(* PLC project FiveDofPlatform.project, CODESYS CODESYS V3.5 SP20 Patch 4 *)
(* stored: creationDateTime 2026-07-31T18:59:57.8348108, modificationDateTime 2026-07-31T18:56:30.8160222 *)

TYPE Axis : STRUCT
  Control_Mode : INT := 0;
  AxisEnable : BOOL;
  伺服绝对位置执行 : MC_MoveAbsolute;  (* 使用实际的功能块类型 *)
  AxisDone : BOOL;
  AxisBusy : BOOL;
  AxisError : BOOL;
  NeedMoveAxis : BOOL := FALSE;
  TargetVel : LREAL;
  TargetAngle : LREAL;
  TargetTorque : LREAL;
  ActualVel : LREAL;
  ActualAngle : LREAL;
  ActualTorque : LREAL;
  AxisLead : LREAL;
  AxisTravel : LREAL;
  AxisGearRatio : LREAL;
  InitDone : BOOL;
  TrigMove : INT;
  StopRequest : BOOL;
  AxisModeSwitchDone : BOOL;
END_STRUCT;
END_TYPE

TYPE LogEntry : STRUCT
  sMessage : STRING(100);  (* 日志内容 *)
  timestamp : DWORD;  (* 时间戳（例如毫秒） *)
  length : WORD;  (* 实际字符串长度 *)
END_STRUCT;
END_TYPE

TYPE LogBuffer : STRUCT
  entries : ARRAY[0..49] OF LogEntry;  (* 50条日志（索引0~49） *)
  writeIdx : INT;  (* 写入位置 (0~49) *)
  readIdx : INT;  (* 已读位置 *)
  count : INT;  (* 未读日志条数 (0~50) *)
  maxSize : INT := 50;  (* 缓冲区容量，固定50 *)
END_STRUCT;
END_TYPE

TYPE LogQueueEntry : STRUCT
  sMsg : STRING(100);
  timestamp : DWORD;
END_STRUCT;
END_TYPE

PROGRAM AxisStatusFeedback_PRG
  VAR
    fbStatusX : Sm3_Basic.MC_ReadStatus;
    fbAxisErrorX : Sm3_Basic.MC_ReadAxisError;
    fbStatusY : Sm3_Basic.MC_ReadStatus;
    fbAxisErrorY : Sm3_Basic.MC_ReadAxisError;
    fbStatusZ : Sm3_Basic.MC_ReadStatus;
    fbAxisErrorZ : Sm3_Basic.MC_ReadAxisError;
    fbStatusB : Sm3_Basic.MC_ReadStatus;
    fbAxisErrorB : Sm3_Basic.MC_ReadAxisError;
    fbStatusC : Sm3_Basic.MC_ReadStatus;
    fbAxisErrorC : Sm3_Basic.MC_ReadAxisError;
    wStatusX : WORD;
    wStatusY : WORD;
    wStatusZ : WORD;
    wStatusB : WORD;
    wStatusC : WORD;
    dwAxisErrorX : DWORD;
    dwAxisErrorY : DWORD;
    dwAxisErrorZ : DWORD;
    dwAxisErrorB : DWORD;
    dwAxisErrorC : DWORD;
    bStatusErrorX : BOOL;
    bStatusFBErrorX : BOOL;
    bStatusAxisErrorX : BOOL;
    bAxisErrorX : BOOL;
    bSwEndSwitchX : BOOL;
    bStatusErrorY : BOOL;
    bStatusFBErrorY : BOOL;
    bStatusAxisErrorY : BOOL;
    bAxisErrorY : BOOL;
    bSwEndSwitchY : BOOL;
    bStatusErrorZ : BOOL;
    bStatusFBErrorZ : BOOL;
    bStatusAxisErrorZ : BOOL;
    bAxisErrorZ : BOOL;
    bSwEndSwitchZ : BOOL;
    bStatusErrorB : BOOL;
    bStatusFBErrorB : BOOL;
    bStatusAxisErrorB : BOOL;
    bAxisErrorB : BOOL;
    bSwEndSwitchB : BOOL;
    bStatusErrorC : BOOL;
    bStatusFBErrorC : BOOL;
    bStatusAxisErrorC : BOOL;
    bAxisErrorC : BOOL;
    bSwEndSwitchC : BOOL;
  END_VAR

            
fbStatusX(
    Axis := AXIS_X,
    Enable := TRUE,
    Valid => ,
    Busy => ,
    Error => bStatusErrorX,
    ErrorID => ,
    Disabled => ,
    Errorstop => ,
    Stopping => ,
    StandStill => ,
    DiscreteMotion => ,
    ContinuousMotion => ,
    SynchronizedMotion => ,
    Homing => ,
    ConstantVelocity => ,
    Accelerating => ,
    Decelerating => ,
    FBErrorOccured => bStatusFBErrorX,
    AxisError => bStatusAxisErrorX
);

fbAxisErrorX(
    Axis := AXIS_X,
    Enable := TRUE,
    Valid => ,
    Busy => ,
    Error => ,
    ErrorID => ,
    AxisError => bAxisErrorX,
    AxisErrorID => dwAxisErrorX,
    SWEndSwitchActive => bSwEndSwitchX
);
IF NOT bAxisErrorX THEN
    dwAxisErrorX := DWORD#0;
END_IF;

wStatusX := WORD#0;
IF fbStatusX.Disabled THEN wStatusX := wStatusX OR WORD#16#0001; END_IF;
IF fbStatusX.Errorstop THEN wStatusX := wStatusX OR WORD#16#0002; END_IF;
IF fbStatusX.Stopping THEN wStatusX := wStatusX OR WORD#16#0004; END_IF;
IF fbStatusX.StandStill THEN wStatusX := wStatusX OR WORD#16#0008; END_IF;
IF fbStatusX.DiscreteMotion THEN wStatusX := wStatusX OR WORD#16#0010; END_IF;
IF fbStatusX.ContinuousMotion THEN wStatusX := wStatusX OR WORD#16#0020; END_IF;
IF fbStatusX.SynchronizedMotion THEN wStatusX := wStatusX OR WORD#16#0040; END_IF;
IF fbStatusX.Homing THEN wStatusX := wStatusX OR WORD#16#0080; END_IF;
IF fbStatusX.ConstantVelocity THEN wStatusX := wStatusX OR WORD#16#0100; END_IF;
IF fbStatusX.Accelerating THEN wStatusX := wStatusX OR WORD#16#0200; END_IF;
IF fbStatusX.Decelerating THEN wStatusX := wStatusX OR WORD#16#0400; END_IF;
IF bStatusErrorX THEN wStatusX := wStatusX OR WORD#16#0800; END_IF;
IF bStatusFBErrorX THEN wStatusX := wStatusX OR WORD#16#1000; END_IF;
IF bStatusAxisErrorX THEN wStatusX := wStatusX OR WORD#16#2000; END_IF;
IF bAxisErrorX THEN wStatusX := wStatusX OR WORD#16#4000; END_IF;
IF bSwEndSwitchX THEN wStatusX := wStatusX OR WORD#16#8000; END_IF;
arReg_data[16] := WORD_TO_INT(wStatusX);
arReg_data[22] := WORD_TO_INT(DWORD_TO_WORD(dwAxisErrorX));
arReg_data[23] := WORD_TO_INT(DWORD_TO_WORD(SHR(dwAxisErrorX, 16)));

fbStatusY(
    Axis := AXIS_Y,
    Enable := TRUE,
    Valid => ,
    Busy => ,
    Error => bStatusErrorY,
    ErrorID => ,
    Disabled => ,
    Errorstop => ,
    Stopping => ,
    StandStill => ,
    DiscreteMotion => ,
    ContinuousMotion => ,
    SynchronizedMotion => ,
    Homing => ,
    ConstantVelocity => ,
    Accelerating => ,
    Decelerating => ,
    FBErrorOccured => bStatusFBErrorY,
    AxisError => bStatusAxisErrorY
);

fbAxisErrorY(
    Axis := AXIS_Y,
    Enable := TRUE,
    Valid => ,
    Busy => ,
    Error => ,
    ErrorID => ,
    AxisError => bAxisErrorY,
    AxisErrorID => dwAxisErrorY,
    SWEndSwitchActive => bSwEndSwitchY
);
IF NOT bAxisErrorY THEN
    dwAxisErrorY := DWORD#0;
END_IF;

wStatusY := WORD#0;
IF fbStatusY.Disabled THEN wStatusY := wStatusY OR WORD#16#0001; END_IF;
IF fbStatusY.Errorstop THEN wStatusY := wStatusY OR WORD#16#0002; END_IF;
IF fbStatusY.Stopping THEN wStatusY := wStatusY OR WORD#16#0004; END_IF;
IF fbStatusY.StandStill THEN wStatusY := wStatusY OR WORD#16#0008; END_IF;
IF fbStatusY.DiscreteMotion THEN wStatusY := wStatusY OR WORD#16#0010; END_IF;
IF fbStatusY.ContinuousMotion THEN wStatusY := wStatusY OR WORD#16#0020; END_IF;
IF fbStatusY.SynchronizedMotion THEN wStatusY := wStatusY OR WORD#16#0040; END_IF;
IF fbStatusY.Homing THEN wStatusY := wStatusY OR WORD#16#0080; END_IF;
IF fbStatusY.ConstantVelocity THEN wStatusY := wStatusY OR WORD#16#0100; END_IF;
IF fbStatusY.Accelerating THEN wStatusY := wStatusY OR WORD#16#0200; END_IF;
IF fbStatusY.Decelerating THEN wStatusY := wStatusY OR WORD#16#0400; END_IF;
IF bStatusErrorY THEN wStatusY := wStatusY OR WORD#16#0800; END_IF;
IF bStatusFBErrorY THEN wStatusY := wStatusY OR WORD#16#1000; END_IF;
IF bStatusAxisErrorY THEN wStatusY := wStatusY OR WORD#16#2000; END_IF;
IF bAxisErrorY THEN wStatusY := wStatusY OR WORD#16#4000; END_IF;
IF bSwEndSwitchY THEN wStatusY := wStatusY OR WORD#16#8000; END_IF;
arReg_data[17] := WORD_TO_INT(wStatusY);
arReg_data[24] := WORD_TO_INT(DWORD_TO_WORD(dwAxisErrorY));
arReg_data[25] := WORD_TO_INT(DWORD_TO_WORD(SHR(dwAxisErrorY, 16)));

fbStatusZ(
    Axis := AXIS_Z,
    Enable := TRUE,
    Valid => ,
    Busy => ,
    Error => bStatusErrorZ,
    ErrorID => ,
    Disabled => ,
    Errorstop => ,
    Stopping => ,
    StandStill => ,
    DiscreteMotion => ,
    ContinuousMotion => ,
    SynchronizedMotion => ,
    Homing => ,
    ConstantVelocity => ,
    Accelerating => ,
    Decelerating => ,
    FBErrorOccured => bStatusFBErrorZ,
    AxisError => bStatusAxisErrorZ
);

fbAxisErrorZ(
    Axis := AXIS_Z,
    Enable := TRUE,
    Valid => ,
    Busy => ,
    Error => ,
    ErrorID => ,
    AxisError => bAxisErrorZ,
    AxisErrorID => dwAxisErrorZ,
    SWEndSwitchActive => bSwEndSwitchZ
);
IF NOT bAxisErrorZ THEN
    dwAxisErrorZ := DWORD#0;
END_IF;

wStatusZ := WORD#0;
IF fbStatusZ.Disabled THEN wStatusZ := wStatusZ OR WORD#16#0001; END_IF;
IF fbStatusZ.Errorstop THEN wStatusZ := wStatusZ OR WORD#16#0002; END_IF;
IF fbStatusZ.Stopping THEN wStatusZ := wStatusZ OR WORD#16#0004; END_IF;
IF fbStatusZ.StandStill THEN wStatusZ := wStatusZ OR WORD#16#0008; END_IF;
IF fbStatusZ.DiscreteMotion THEN wStatusZ := wStatusZ OR WORD#16#0010; END_IF;
IF fbStatusZ.ContinuousMotion THEN wStatusZ := wStatusZ OR WORD#16#0020; END_IF;
IF fbStatusZ.SynchronizedMotion THEN wStatusZ := wStatusZ OR WORD#16#0040; END_IF;
IF fbStatusZ.Homing THEN wStatusZ := wStatusZ OR WORD#16#0080; END_IF;
IF fbStatusZ.ConstantVelocity THEN wStatusZ := wStatusZ OR WORD#16#0100; END_IF;
IF fbStatusZ.Accelerating THEN wStatusZ := wStatusZ OR WORD#16#0200; END_IF;
IF fbStatusZ.Decelerating THEN wStatusZ := wStatusZ OR WORD#16#0400; END_IF;
IF bStatusErrorZ THEN wStatusZ := wStatusZ OR WORD#16#0800; END_IF;
IF bStatusFBErrorZ THEN wStatusZ := wStatusZ OR WORD#16#1000; END_IF;
IF bStatusAxisErrorZ THEN wStatusZ := wStatusZ OR WORD#16#2000; END_IF;
IF bAxisErrorZ THEN wStatusZ := wStatusZ OR WORD#16#4000; END_IF;
IF bSwEndSwitchZ THEN wStatusZ := wStatusZ OR WORD#16#8000; END_IF;
arReg_data[18] := WORD_TO_INT(wStatusZ);
arReg_data[26] := WORD_TO_INT(DWORD_TO_WORD(dwAxisErrorZ));
arReg_data[27] := WORD_TO_INT(DWORD_TO_WORD(SHR(dwAxisErrorZ, 16)));

fbStatusB(
    Axis := AXIS_B,
    Enable := TRUE,
    Valid => ,
    Busy => ,
    Error => bStatusErrorB,
    ErrorID => ,
    Disabled => ,
    Errorstop => ,
    Stopping => ,
    StandStill => ,
    DiscreteMotion => ,
    ContinuousMotion => ,
    SynchronizedMotion => ,
    Homing => ,
    ConstantVelocity => ,
    Accelerating => ,
    Decelerating => ,
    FBErrorOccured => bStatusFBErrorB,
    AxisError => bStatusAxisErrorB
);

fbAxisErrorB(
    Axis := AXIS_B,
    Enable := TRUE,
    Valid => ,
    Busy => ,
    Error => ,
    ErrorID => ,
    AxisError => bAxisErrorB,
    AxisErrorID => dwAxisErrorB,
    SWEndSwitchActive => bSwEndSwitchB
);
IF NOT bAxisErrorB THEN
    dwAxisErrorB := DWORD#0;
END_IF;

wStatusB := WORD#0;
IF fbStatusB.Disabled THEN wStatusB := wStatusB OR WORD#16#0001; END_IF;
IF fbStatusB.Errorstop THEN wStatusB := wStatusB OR WORD#16#0002; END_IF;
IF fbStatusB.Stopping THEN wStatusB := wStatusB OR WORD#16#0004; END_IF;
IF fbStatusB.StandStill THEN wStatusB := wStatusB OR WORD#16#0008; END_IF;
IF fbStatusB.DiscreteMotion THEN wStatusB := wStatusB OR WORD#16#0010; END_IF;
IF fbStatusB.ContinuousMotion THEN wStatusB := wStatusB OR WORD#16#0020; END_IF;
IF fbStatusB.SynchronizedMotion THEN wStatusB := wStatusB OR WORD#16#0040; END_IF;
IF fbStatusB.Homing THEN wStatusB := wStatusB OR WORD#16#0080; END_IF;
IF fbStatusB.ConstantVelocity THEN wStatusB := wStatusB OR WORD#16#0100; END_IF;
IF fbStatusB.Accelerating THEN wStatusB := wStatusB OR WORD#16#0200; END_IF;
IF fbStatusB.Decelerating THEN wStatusB := wStatusB OR WORD#16#0400; END_IF;
IF bStatusErrorB THEN wStatusB := wStatusB OR WORD#16#0800; END_IF;
IF bStatusFBErrorB THEN wStatusB := wStatusB OR WORD#16#1000; END_IF;
IF bStatusAxisErrorB THEN wStatusB := wStatusB OR WORD#16#2000; END_IF;
IF bAxisErrorB THEN wStatusB := wStatusB OR WORD#16#4000; END_IF;
IF bSwEndSwitchB THEN wStatusB := wStatusB OR WORD#16#8000; END_IF;
arReg_data[20] := WORD_TO_INT(wStatusB);
arReg_data[28] := WORD_TO_INT(DWORD_TO_WORD(dwAxisErrorB));
arReg_data[29] := WORD_TO_INT(DWORD_TO_WORD(SHR(dwAxisErrorB, 16)));

fbStatusC(
    Axis := AXIS_C,
    Enable := TRUE,
    Valid => ,
    Busy => ,
    Error => bStatusErrorC,
    ErrorID => ,
    Disabled => ,
    Errorstop => ,
    Stopping => ,
    StandStill => ,
    DiscreteMotion => ,
    ContinuousMotion => ,
    SynchronizedMotion => ,
    Homing => ,
    ConstantVelocity => ,
    Accelerating => ,
    Decelerating => ,
    FBErrorOccured => bStatusFBErrorC,
    AxisError => bStatusAxisErrorC
);

fbAxisErrorC(
    Axis := AXIS_C,
    Enable := TRUE,
    Valid => ,
    Busy => ,
    Error => ,
    ErrorID => ,
    AxisError => bAxisErrorC,
    AxisErrorID => dwAxisErrorC,
    SWEndSwitchActive => bSwEndSwitchC
);
IF NOT bAxisErrorC THEN
    dwAxisErrorC := DWORD#0;
END_IF;

wStatusC := WORD#0;
IF fbStatusC.Disabled THEN wStatusC := wStatusC OR WORD#16#0001; END_IF;
IF fbStatusC.Errorstop THEN wStatusC := wStatusC OR WORD#16#0002; END_IF;
IF fbStatusC.Stopping THEN wStatusC := wStatusC OR WORD#16#0004; END_IF;
IF fbStatusC.StandStill THEN wStatusC := wStatusC OR WORD#16#0008; END_IF;
IF fbStatusC.DiscreteMotion THEN wStatusC := wStatusC OR WORD#16#0010; END_IF;
IF fbStatusC.ContinuousMotion THEN wStatusC := wStatusC OR WORD#16#0020; END_IF;
IF fbStatusC.SynchronizedMotion THEN wStatusC := wStatusC OR WORD#16#0040; END_IF;
IF fbStatusC.Homing THEN wStatusC := wStatusC OR WORD#16#0080; END_IF;
IF fbStatusC.ConstantVelocity THEN wStatusC := wStatusC OR WORD#16#0100; END_IF;
IF fbStatusC.Accelerating THEN wStatusC := wStatusC OR WORD#16#0200; END_IF;
IF fbStatusC.Decelerating THEN wStatusC := wStatusC OR WORD#16#0400; END_IF;
IF bStatusErrorC THEN wStatusC := wStatusC OR WORD#16#0800; END_IF;
IF bStatusFBErrorC THEN wStatusC := wStatusC OR WORD#16#1000; END_IF;
IF bStatusAxisErrorC THEN wStatusC := wStatusC OR WORD#16#2000; END_IF;
IF bAxisErrorC THEN wStatusC := wStatusC OR WORD#16#4000; END_IF;
IF bSwEndSwitchC THEN wStatusC := wStatusC OR WORD#16#8000; END_IF;
arReg_data[21] := WORD_TO_INT(wStatusC);
arReg_data[30] := WORD_TO_INT(DWORD_TO_WORD(dwAxisErrorC));
arReg_data[31] := WORD_TO_INT(DWORD_TO_WORD(SHR(dwAxisErrorC, 16)));
            
          
END_PROGRAM

PROGRAM Axis_Y_PRG
  VAR
    伺服使能 : Sm3_Basic.MC_Power;  (* 轴功能块实例 *)
    伺服绝对位置执行 : Sm3_Basic.MC_MoveAbsolute;
    伺服实际位置 : Sm3_Basic.MC_ReadActualPosition;
    伺服停止 : Sm3_Basic.MC_Stop;
    伺服复位 : Sm3_Basic.MC_Reset;
    伺服状态 : Sm3_Basic.MC_ReadStatus;
    复位轴组 : Sm3_Basic.SMC3_ReinitDrive;
    当前位置 : LREAL;  (* 变量 *)
    轴组复位 : BOOL;
    目标位置 : LREAL;
    目标速度 : LREAL;
    伺服错误状态 : BOOL;
    轴使能状态 : BOOL;
    总线状态 : BOOL;
    复位触发 : R_TRIG;  (* 报警清除相关 *)
    复位请求 : BOOL;
    复位中 : BOOL;
    POS_DEAD_ZONE : REAL := 0.01;  (* 死区常量 *)
    伺服复位_Done : BOOL;
    debug_Done_Status : BOOL;  (* 在 AXIS_Y0_PRG 中添加 *)
    debug_KeepEnable : BOOL;
    move_trigger : R_TRIG;  (* 脉冲触发相关 *)
    AXIS_Y_EXCUSE : BOOL := FALSE;
    log_msg : STRING(100);
  END_VAR

                    //------------------------------------------------------------------
// Z 轴控制逻辑（简化版 - 仅上升沿触发）
//------------------------------------------------------------------

// 读取实际位置
伺服实际位置(
    Axis    := AXIS_Y,
    Enable  := TRUE,
    Position=> 当前位置
);
GVL.Axes[2].ActualAngle := 当前位置;

// 读取轴状态
伺服状态(
    Axis    := AXIS_Y,
    Enable  := TRUE,
    Valid   => ,
    Busy    => ,
    Error   => 伺服错误状态,
    ErrorID => ,
    Disabled=> 总线状态
);

// 轴使能控制
伺服使能(
    Axis               := AXIS_Y,
    Enable             := TRUE,
    bRegulatorOn       := GVL.Axes[2].AxisEnable,
    bDriveStart        := GVL.Axes[2].AxisEnable,
    Status             => 轴使能状态,
    bRegulatorRealState=> ,
    bDriveStartRealState=> ,
    Busy               => ,
    Error              => ,
    ErrorID            =>
);

// 目标位置、速度赋值（来自全局变量）
目标位置 := GVL.Axes[2].TargetAngle;
目标速度 :=  GVL.Axes[2].TargetVel;

// ********** 核心：上升沿触发运动 **********
// 使用 R_TRIG 检测 need_move 的上升沿
move_trigger(CLK := GVL.Axes[2].NeedMoveAxis);
IF move_trigger.Q THEN
    AXIS_Y_EXCUSE := TRUE;   // 产生一个扫描周期的脉冲
	log_msg := 'X-axis has been triggered';
// 	logfb(write:=TRUE,sFileTestString:=log_msg);
	AppendLog(log_msg);
ELSE
    AXIS_Y_EXCUSE := FALSE;
END_IF

// 绝对定位指令
GVL.Axes[2].伺服绝对位置执行(
    Axis        := AXIS_Y,
    Execute     := AXIS_Y_EXCUSE,
    Position    := 目标位置,
    Velocity    := 目标速度,
    Acceleration:= 10000,//4000  //85000
    Deceleration:= 10000,//4000  //85000
    Jerk        := ,
    Direction   := ,
    BufferMode  := ,
    Done        => GVL.Axes[2].InitDone,
    Busy        => ,
    Active      => ,
    CommandAborted=> ,
    Error       => GVL.Axes[2].AxisError,
    ErrorID     =>
);

// 运动完成：清除 need_move 并通知状态机
IF  GVL.Axes[2].InitDone THEN
    GVL.Axes[2].NeedMoveAxis := FALSE;              // 清除运动请求
    GVL.Axes[2].AxisDone := TRUE;         // 通知状态机运动完成
	log_msg := 'X-Axis movement completed! ';
// 	logfb(write:=TRUE,sFileTestString:=log_msg);
// 	AppendLog(log_msg);
END_IF

// 复位功能块（保持不变）
伺服复位(
    Axis    := AXIS_Y,
    Execute := 复位中 AND NOT 伺服复位.Done,
    Done    => ,
    Busy    => ,
    Error   => ,
    ErrorID =>
);

复位轴组(
    Axis      := AXIS_Y,
    bExecute  := 伺服复位.Done,
    bVirtual  := FALSE,
    bDone     => ,
    bBusy     => ,
    bError    => ,
    nErrorID  =>
);

// 报警清除逻辑
复位触发(CLK := (伺服错误状态 OR 复位请求) AND NOT 复位中);
IF 复位触发.Q THEN
    复位中 := TRUE;
    复位请求 := FALSE;
END_IF

IF 伺服复位.Done THEN
    复位中 := FALSE;
END_IF
                  
END_PROGRAM

PROGRAM ModbusTcpSlave
  VAR CONSTANT
    aAngleFactor : ARRAY[1..GVL.AXIS_COUNT] OF REAL := [(360.0 / 26.0), (360.0 / 5.0), (360.0 / 5.0), 1, 1];
  END_VAR
  VAR
    modTcpSlaveInit : gcan.FB_ModbusTCP_Slave_Init;  (* Modbus TCP Slave初始化功能块 *)
    modTcpSlaveCtrl : gcan.FB_ModbusTCP_Slave_Ctrl;  (* Modbus TCP Slave执行功能块 *)
    eout : BOOL;  (* 用于承接功能块中完成标志引脚数据的变量 *)
    iSocket : INT;  (* 用于存放自身socket *)
    uiErr : UINT;  (* 用于承接功能块中报错引脚错误信息的变量 *)
    isInit : BOOL := FALSE;  (* 用于初始化执行一次的逻辑变量 *)
    arClient : ARRAY[0..10] OF INT;  (* 用于存放Client即主站的socket *)
    btargetAngleChange : BOOL := FALSE;
    OldTargetAngle : WORD;
    enCtr : BOOL := FALSE;  (* Modbus TCP Slave执行功能块使能变量 *)
    iTemp : INT;  (* 临时变量，用于32位数据转换 *)
    dwAngle : INT;  (* 32位临时存储，用于组合角度寄存器 *)
    i : INT;
    wTemp : WORD;  (* modbuslog *)
    sCurLog : STRING(100);
    iLen : INT;
    pCurEntry : POINTER TO LogEntry;
    iCharIdx : INT;
    iRegIdx : INT;
  END_VAR

                    // ================================
// 日志映射部分：将当前未读日志填充到保持寄存器
// ================================
IF g_LogBuffer.count > 0 THEN
    // 获取当前读指针指向的日志条目
    pCurEntry := ADR(g_LogBuffer.entries[g_LogBuffer.readIdx]);
    sCurLog := pCurEntry^.sMessage;
    iLen := pCurEntry^.length;
    
    // 地址100：日志长度（WORD）
    arReg_data[100] := INT_TO_WORD(iLen);
    
    // 地址101-102：时间戳（低字，高字）
    arReg_data[101] := DWORD_TO_WORD(pCurEntry^.timestamp AND 16#FFFF);
    arReg_data[102] := DWORD_TO_WORD(SHR(pCurEntry^.timestamp, 16));
    
    // 清空字符串缓冲区寄存器（地址103 ~ 152，共50个WORD）
    FOR i := 103 TO 152 DO
        arReg_data[i] := 0;
    END_FOR
    
    // ----- 将字符串每两个字符打包成一个 WORD -----
    // 注意：你的环境中字符串索引从0开始（已验证）
    iCharIdx := 0;      // 当前字符索引（从0开始）
    iRegIdx := 103;     // 当前寄存器地址
    WHILE iCharIdx < iLen DO
        // 低字节 = 第一个字符
        wTemp := sCurLog[iCharIdx];
        iCharIdx := iCharIdx + 1;
        // 如果有下一个字符，放入高字节
        IF iCharIdx < iLen THEN
            wTemp := wTemp OR SHL(sCurLog[iCharIdx], 8);
            iCharIdx := iCharIdx + 1;
        END_IF
        arReg_data[iRegIdx] := wTemp;
        iRegIdx := iRegIdx + 1;
    END_WHILE
ELSE
    // 无未读日志，长度寄存器写0
    arReg_data[100] := 0;
END_IF

// --------------------------------
// 处理主站确认线圈（地址16）
// --------------------------------
IF arDo_data[16] THEN
    IF g_LogBuffer.count > 0 THEN
        g_LogBuffer.readIdx := (g_LogBuffer.readIdx + 1) MOD g_LogBuffer.maxSize;
        g_LogBuffer.count := g_LogBuffer.count - 1;
    END_IF
    arDo_data[16] := FALSE;
END_IF





IF isInit=FALSE THEN							

	modtcpslaveinit(en_in:=TRUE,					//Modbus TCP Slave初始化功能块使能
	xenable:=TRUE,									//使能初始化功能
	iport:=502,										//开放端口号502
	en_out=>eout,									//Modbus TCP Slave初始化功能块执行完成
	isocket=>iSocket,								//创建的socket存入变量
	uierror=>uiErr);								//Modbus TCP Slave初始化功能块执行错误信息
	
	IF isocket>=0 AND uiErr=0 THEN					//成功创建socket且无错误，逻辑标志置位，下周期执行ELSE
		isInit:=TRUE;	
		
		enCtr:=FALSE;
		ELSE                                        //等待连接成功
		modtcpslaveinit(en_in:=0,xenable:=0);	
	END_IF
 
ELSE


	// 循环读取电机位置
	FOR i := 1 TO GVL.AXIS_COUNT DO
		arAi_data[i] := INT_TO_WORD(REAL_TO_INT(Axes[i].ActualAngle/aAngleFactor[i]*10.0));
	END_FOR
	Move_5Axis_Sign:=arReg_data[0];
	
	
	// 循环处理前7个通道（目标角度数组）
	IF 	bfiveDOF_state =0 THEN
		FOR i := 1 TO GVL.AXIS_COUNT DO
			dwAngle := WORD_TO_INT(arReg_data[i]);      // 有符号原始值
			PlatformTargetAngle[i] := dwAngle * aAngleFactor[i];
		END_FOR

	END_IF
  xJogMode[1] := (arReg_data[19] AND WORD#16#0001) <> WORD#0; // X
  xJogMode[2] := (arReg_data[19] AND WORD#16#0002) <> WORD#0; // Y
  xJogMode[3] := (arReg_data[19] AND WORD#16#0004) <> WORD#0; // Z
  xJogMode[4] := (arReg_data[19] AND WORD#16#0008) <> WORD#0; // B
  xJogMode[5] := (arReg_data[19] AND WORD#16#0010) <> WORD#0; // C
  
  xJogFwd[1] := xJogMode[1] AND (arReg_data[6] <> WORD#0);
  xJogRev[1] := xJogMode[1] AND (arReg_data[7] <> WORD#0);

  xJogFwd[2] := xJogMode[2] AND (arReg_data[8] <> WORD#0);
  xJogRev[2] := xJogMode[2] AND (arReg_data[9] <> WORD#0);

  xJogFwd[3] := xJogMode[3] AND (arReg_data[10] <> WORD#0);
  xJogRev[3] := xJogMode[3] AND (arReg_data[11] <> WORD#0);

  xJogFwd[4] := xJogMode[4] AND (arReg_data[12] <> WORD#0);
  xJogRev[4] := xJogMode[4] AND (arReg_data[13] <> WORD#0);

  xJogFwd[5] := xJogMode[5] AND (arReg_data[14] <> WORD#0);
  xJogRev[5] := xJogMode[5] AND (arReg_data[15] <> WORD#0);
  
  xJogFwd[1] := arReg_data[6] <> 0;
  xJogRev[1] := arReg_data[7] <> 0;

  xJogFwd[2] := arReg_data[8] <> 0;
  xJogRev[2] := arReg_data[9] <> 0;

  xJogFwd[3] := arReg_data[10] <> 0;
  xJogRev[3] := arReg_data[11] <> 0;

  xJogFwd[4] := arReg_data[12] <> 0;
  xJogRev[4] := arReg_data[13] <> 0;

  xJogFwd[5] := arReg_data[14] <> 0;
  xJogRev[5] := arReg_data[15] <> 0;

	modtcpslavectrl(en_in:=enCtr,					//Modbus TCP Slave执行功能块使能
	xenable:=TRUE,									//Modbus TCP Slave执行功能使能
	isocket:=isocket,								//输入创建的socket
	dwatchdogtime:=2000,							//看门狗时间
	p_clientsocket:=ADR(arClient),					//将连接进来的socket存放到数组
	imaxclientcount:=10,							//设置最大连接数量
	uido_number:=17,uido_startaddr:=0,pdo_data:=ADR(arDo_data),		//uido_number设定线圈个数，uido_startaddr设定线圈起始地址，数据存放在arDo_data数组
	uidi_number:=16,uidi_startaddr:=0,pdi_data:=ADR(arDi_data),		//uidi_number设定离散型数据个数，uidi_startaddr设定离散型数据起始地址，数据存放在arDi_data数组
	uireg_number:=200,uireg_startaddr:=0,preg_data:=ADR(arReg_data), //uireg_number设定保持型寄存器个数，uireg_startaddr设定保持型寄存器起始地址，数据存放在arReg_data数组
	uiai_number:=16,uiai_startaddr:=0,pai_data:=ADR(arAi_data),		//uiai_number设定输入型寄存器个数，uiai_startaddr设定输入型寄存器起始地址，数据存放在arAi_data数组
	en_out=>eout,									//Modbus TCP Slave执行功能块执行完成
	uierror=>uierr);								//Modbus TCP Slave执行功能块执行错误信息
	enctr:=TRUE;
	IF uierr <>0 THEN                               //如果从站报错，则重新连接从站
		modtcpslaveinit(en_in:=0,xenable:=0);	
		isInit:=0;
	END_IF
END_IF

 
// 释放锁
g_LogLock := FALSE;
 
                  
END_PROGRAM

PROGRAM PLC_PRG
  VAR
    startMove : BOOL;
    platTargetangle : ARRAY[1..7] OF LREAL;
    platTargetvel : ARRAY[1..7] OF LREAL;
    fbMove6DOF : FB_5DOF_Platform_Move;
    iAxis : INT;
    MaxVel : UDINT := 2048576000;
    bcontrol : UINT;
    logfb : Syslog_FB;
    log_msg : STRING(100);
  END_VAR

                    
                  
END_PROGRAM

FUNCTION_BLOCK FB_5DOF_Platform_Move
  VAR_IN_OUT
    AxisAngle : ARRAY[1..AXIS_COUNT] OF LREAL;
    AxisVel : ARRAY[1..AXIS_COUNT] OF LREAL;
  END_VAR
  VAR_INPUT
    Execute : BOOL;
    Monitor : BOOL;
  END_VAR
  VAR_OUTPUT
    Done : BOOL;
    Busy : BOOL;
    Error : BOOL;
    ErrorID : WORD;
  END_VAR
  VAR
    trigExec : R_TRIG;
    xInternal : BOOL;
    i : INT;
    allDone : BOOL := FALSE;
    anyError : BOOL;
    errId : WORD;
  END_VAR

                    
// 上升沿触发：锁存目标值并开始运动
trigExec(CLK := Execute);
IF trigExec.Q THEN
    FOR i := 1 TO AXIS_COUNT DO
        GVL.Axes[i].TargetAngle := AxisAngle[i];
		GVL.Axes[i].TargetVel:=AxisVel[i];
    END_FOR
//     xInternal := TRUE;
    Busy := TRUE;
    Done := FALSE;
    Error := FALSE;
    ErrorID := 0;
END_IF

// 监控所有轴的状态（需要你的单轴功能块实例：AXIS_X伺服绝对位置执行 等）
IF Monitor  THEN
    allDone := TRUE;
    anyError := FALSE;
    errId := 0;
    
    // 检查每个轴（请根据实际轴名修改，以下为示例）
	FOR i :=1 TO AXIS_COUNT DO
		IF NOT GVL.Axes[i].AxisDone THEN allDone := FALSE; END_IF
		IF GVL.Axes[i].AxisError THEN anyError := TRUE; errId := GVL.Axes[i].伺服绝对位置执行.ErrorID; END_IF
	END_FOR
  
    
    IF  allDone THEN
        Busy := FALSE;
        Done := TRUE;
        xInternal := FALSE;
    END_IF
END_IF
                  
END_FUNCTION_BLOCK

PROGRAM AXIS_X_PRG
  VAR
    伺服使能 : Sm3_Basic.MC_Power;  (* 轴功能块实例 *)
    伺服绝对位置执行 : Sm3_Basic.MC_MoveAbsolute;
    伺服实际位置 : Sm3_Basic.MC_ReadActualPosition;
    伺服停止 : Sm3_Basic.MC_Stop;
    伺服复位 : Sm3_Basic.MC_Reset;
    伺服状态 : Sm3_Basic.MC_ReadStatus;
    复位轴组 : Sm3_Basic.SMC3_ReinitDrive;
    当前位置 : LREAL;  (* 变量 *)
    轴组复位 : BOOL;
    目标位置 : LREAL;
    目标速度 : LREAL;
    伺服错误状态 : BOOL;
    轴使能状态 : BOOL;
    总线状态 : BOOL;
    复位触发 : R_TRIG;  (* 报警清除相关 *)
    复位请求 : BOOL;
    复位中 : BOOL;
    POS_DEAD_ZONE : REAL := 0.01;  (* 死区常量 *)
    move_trigger : R_TRIG;
    AXIS_X_EXCUSE : BOOL := FALSE;
    log_msg : STRING(100);
  END_VAR

                    //------------------------------------------------------------------
// Z 轴控制逻辑（简化版 - 仅上升沿触发）
//------------------------------------------------------------------

// 读取实际位置
伺服实际位置(
    Axis    := AXIS_X,
    Enable  := TRUE,
    Position=> 当前位置
);
GVL.Axes[1].ActualAngle := 当前位置;

// 读取轴状态
伺服状态(
    Axis    := AXIS_X,
    Enable  := TRUE,
    Valid   => ,
    Busy    => ,
    Error   => 伺服错误状态,
    ErrorID => ,
    Disabled=> 总线状态
);

// 轴使能控制
伺服使能(
    Axis               := AXIS_X,
    Enable             := TRUE,
    bRegulatorOn       := GVL.Axes[1].AxisEnable,
    bDriveStart        := GVL.Axes[1].AxisEnable,
    Status             => 轴使能状态,
    bRegulatorRealState=> ,
    bDriveStartRealState=> ,
    Busy               => ,
    Error              => ,
    ErrorID            =>
);

// 目标位置、速度赋值（来自全局变量）
目标位置 := GVL.Axes[1].TargetAngle;
目标速度 :=  GVL.Axes[1].TargetVel;

// ********** 核心：上升沿触发运动 **********
// 使用 R_TRIG 检测 need_move 的上升沿
move_trigger(CLK := GVL.Axes[1].NeedMoveAxis);
IF move_trigger.Q THEN
    AXIS_X_EXCUSE := TRUE;   // 产生一个扫描周期的脉冲
	log_msg := 'X-axis has been triggered';
// 	logfb(write:=TRUE,sFileTestString:=log_msg);
	AppendLog(log_msg);
ELSE
    AXIS_X_EXCUSE := FALSE;
END_IF

// 绝对定位指令
GVL.Axes[1].伺服绝对位置执行(
    Axis        := AXIS_X,
    Execute     := AXIS_X_EXCUSE,
    Position    := 目标位置,
    Velocity    := 目标速度,
    Acceleration:= 10000,//4000  //85000
    Deceleration:= 10000,//4000  //85000
    Jerk        := ,
    Direction   := ,
    BufferMode  := ,
    Done        => GVL.Axes[1].InitDone,
    Busy        => ,
    Active      => ,
    CommandAborted=> ,
    Error       => GVL.Axes[1].AxisError,
    ErrorID     =>
);

// 运动完成：清除 need_move 并通知状态机
IF  GVL.Axes[1].InitDone THEN
    GVL.Axes[1].NeedMoveAxis := FALSE;              // 清除运动请求
    GVL.Axes[1].AxisDone := TRUE;         // 通知状态机运动完成
	log_msg := 'X-Axis movement completed! ';
// 	logfb(write:=TRUE,sFileTestString:=log_msg);
// 	AppendLog(log_msg);
END_IF

// 复位功能块（保持不变）
伺服复位(
    Axis    := AXIS_X,
    Execute := 复位中 AND NOT 伺服复位.Done,
    Done    => ,
    Busy    => ,
    Error   => ,
    ErrorID =>
);

复位轴组(
    Axis      := AXIS_X,
    bExecute  := 伺服复位.Done,
    bVirtual  := FALSE,
    bDone     => ,
    bBusy     => ,
    bError    => ,
    nErrorID  =>
);

// 报警清除逻辑
复位触发(CLK := (伺服错误状态 OR 复位请求) AND NOT 复位中);
IF 复位触发.Q THEN
    复位中 := TRUE;
    复位请求 := FALSE;
END_IF

IF 伺服复位.Done THEN
    复位中 := FALSE;
END_IF
                  
END_PROGRAM

PROGRAM AXIS_B_PRG
  VAR
    伺服使能 : Sm3_Basic.MC_Power;  (* 轴功能块实例 *)
    伺服绝对位置执行 : Sm3_Basic.MC_MoveAbsolute;
    伺服实际位置 : Sm3_Basic.MC_ReadActualPosition;
    伺服停止 : Sm3_Basic.MC_Stop;
    伺服复位 : Sm3_Basic.MC_Reset;
    伺服状态 : Sm3_Basic.MC_ReadStatus;
    复位轴组 : Sm3_Basic.SMC3_ReinitDrive;
    当前位置 : LREAL;  (* 变量 *)
    轴组复位 : BOOL;
    目标位置 : LREAL;
    目标速度 : LREAL;
    伺服错误状态 : BOOL;
    轴使能状态 : BOOL;
    总线状态 : BOOL;
    复位触发 : R_TRIG;  (* 报警清除相关 *)
    复位请求 : BOOL;
    复位中 : BOOL;
    move_trigger : R_TRIG;
    AXIS_B_EXCUSE : BOOL := FALSE;
    log_msg : STRING(100);
  END_VAR

                    //------------------------------------------------------------------
// Z 轴控制逻辑（简化版 - 仅上升沿触发）
//------------------------------------------------------------------

// 读取实际位置
伺服实际位置(
    Axis    := AXIS_B,
    Enable  := TRUE,
    Position=> 当前位置
);
GVL.Axes[4].ActualAngle := 当前位置;

// 读取轴状态
伺服状态(
    Axis    := AXIS_B,
    Enable  := TRUE,
    Valid   => ,
    Busy    => ,
    Error   => 伺服错误状态,
    ErrorID => ,
    Disabled=> 总线状态
);

// 轴使能控制
伺服使能(
    Axis               := AXIS_B,
    Enable             := TRUE,
    bRegulatorOn       := GVL.Axes[4].AxisEnable,
    bDriveStart        := GVL.Axes[4].AxisEnable,
    Status             => 轴使能状态,
    bRegulatorRealState=> ,
    bDriveStartRealState=> ,
    Busy               => ,
    Error              => ,
    ErrorID            =>
);

// 目标位置、速度赋值（来自全局变量）
目标位置 := GVL.Axes[4].TargetAngle;
目标速度 :=  GVL.Axes[4].TargetVel;

// ********** 核心：上升沿触发运动 **********
// 使用 R_TRIG 检测 need_move 的上升沿
move_trigger(CLK := GVL.Axes[4].NeedMoveAxis);
IF move_trigger.Q THEN
    AXIS_B_EXCUSE := TRUE;   // 产生一个扫描周期的脉冲
	log_msg := 'X-axis has been triggered';
// 	logfb(write:=TRUE,sFileTestString:=log_msg);
	AppendLog(log_msg);
ELSE
    AXIS_B_EXCUSE := FALSE;
END_IF

// 绝对定位指令
GVL.Axes[4].伺服绝对位置执行(
    Axis        := AXIS_B,
    Execute     := AXIS_B_EXCUSE,
    Position    := 目标位置,
    Velocity    := 目标速度,
    Acceleration:= 10000,//4000  //85000
    Deceleration:= 10000,//4000  //85000
    Jerk        := ,
    Direction   := ,
    BufferMode  := ,
    Done        => GVL.Axes[4].InitDone,
    Busy        => ,
    Active      => ,
    CommandAborted=> ,
    Error       => GVL.Axes[4].AxisError,
    ErrorID     =>
);

// 运动完成：清除 need_move 并通知状态机
IF  GVL.Axes[4].InitDone THEN
    GVL.Axes[4].NeedMoveAxis := FALSE;              // 清除运动请求
    GVL.Axes[4].AxisDone := TRUE;         // 通知状态机运动完成
	log_msg := 'B-Axis movement completed! ';
// 	logfb(write:=TRUE,sFileTestString:=log_msg);
// 	AppendLog(log_msg);
END_IF

// 复位功能块（保持不变）
伺服复位(
    Axis    := AXIS_B,
    Execute := 复位中 AND NOT 伺服复位.Done,
    Done    => ,
    Busy    => ,
    Error   => ,
    ErrorID =>
);

复位轴组(
    Axis      := AXIS_B,
    bExecute  := 伺服复位.Done,
    bVirtual  := FALSE,
    bDone     => ,
    bBusy     => ,
    bError    => ,
    nErrorID  =>
);

// 报警清除逻辑
复位触发(CLK := (伺服错误状态 OR 复位请求) AND NOT 复位中);
IF 复位触发.Q THEN
    复位中 := TRUE;
    复位请求 := FALSE;
END_IF

IF 伺服复位.Done THEN
    复位中 := FALSE;
END_IF
                  
END_PROGRAM

PROGRAM AXIS_Z_PRG
  VAR
    伺服使能 : Sm3_Basic.MC_Power;  (* 轴功能块实例 *)
    伺服绝对位置执行 : Sm3_Basic.MC_MoveAbsolute;
    伺服实际位置 : Sm3_Basic.MC_ReadActualPosition;
    伺服停止 : Sm3_Basic.MC_Stop;
    伺服复位 : Sm3_Basic.MC_Reset;
    伺服状态 : Sm3_Basic.MC_ReadStatus;
    复位轴组 : Sm3_Basic.SMC3_ReinitDrive;
    当前位置 : LREAL;  (* 变量 *)
    轴组复位 : BOOL;
    目标位置 : LREAL;
    目标速度 : LREAL;
    伺服错误状态 : BOOL;
    轴使能状态 : BOOL;
    总线状态 : BOOL;
    复位触发 : R_TRIG;  (* 报警清除相关 *)
    复位请求 : BOOL;
    复位中 : BOOL;
    伺服复位_Done : BOOL;
    debug_Done_Status : BOOL;  (* 在 AXIS_Z_PRG 中添加 *)
    debug_KeepEnable : BOOL;
    move_trigger : R_TRIG;  (* 脉冲触发相关 *)
    AXIS_Z_EXCUSE : BOOL := FALSE;
    log_msg : STRING(100);
  END_VAR

                    //------------------------------------------------------------------
// Z 轴控制逻辑（简化版 - 仅上升沿触发）
//------------------------------------------------------------------

// 读取实际位置
伺服实际位置(
    Axis    := AXIS_Z,
    Enable  := TRUE,
    Position=> 当前位置
);
GVL.Axes[3].ActualAngle := 当前位置;

// 读取轴状态
伺服状态(
    Axis    := AXIS_Z,
    Enable  := TRUE,
    Valid   => ,
    Busy    => ,
    Error   => 伺服错误状态,
    ErrorID => ,
    Disabled=> 总线状态
);

// 轴使能控制
伺服使能(
    Axis               := AXIS_Z,
    Enable             := TRUE,
    bRegulatorOn       := GVL.Axes[3].AxisEnable,
    bDriveStart        := GVL.Axes[3].AxisEnable,
    Status             => 轴使能状态,
    bRegulatorRealState=> ,
    bDriveStartRealState=> ,
    Busy               => ,
    Error              => ,
    ErrorID            =>
);

// 目标位置、速度赋值（来自全局变量）
目标位置 := GVL.Axes[3].TargetAngle;
目标速度 :=  GVL.Axes[3].TargetVel;

// ********** 核心：上升沿触发运动 **********
// 使用 R_TRIG 检测 need_move 的上升沿
move_trigger(CLK := GVL.Axes[3].NeedMoveAxis);
IF move_trigger.Q THEN
    AXIS_Z_EXCUSE := TRUE;   // 产生一个扫描周期的脉冲
	log_msg := 'X-axis has been triggered';
// 	logfb(write:=TRUE,sFileTestString:=log_msg);
	AppendLog(log_msg);
ELSE
    AXIS_Z_EXCUSE := FALSE;
END_IF

// 绝对定位指令
GVL.Axes[3].伺服绝对位置执行(
    Axis        := AXIS_Z,
    Execute     := AXIS_Z_EXCUSE,
    Position    := 目标位置,
    Velocity    := 目标速度,
    Acceleration:= 10000,//4000  //85000
    Deceleration:= 10000,//4000  //85000
    Jerk        := ,
    Direction   := ,
    BufferMode  := ,
    Done        => GVL.Axes[3].InitDone,
    Busy        => ,
    Active      => ,
    CommandAborted=> ,
    Error       => GVL.Axes[3].AxisError,
    ErrorID     =>
);

// 运动完成：清除 need_move 并通知状态机
IF  GVL.Axes[3].InitDone THEN
    GVL.Axes[3].NeedMoveAxis := FALSE;              // 清除运动请求
    GVL.Axes[3].AxisDone := TRUE;         // 通知状态机运动完成
	log_msg := 'Z-Axis movement completed! ';
// 	logfb(write:=TRUE,sFileTestString:=log_msg);
// 	AppendLog(log_msg);
END_IF

// 复位功能块（保持不变）
伺服复位(
    Axis    := AXIS_Z,
    Execute := 复位中 AND NOT 伺服复位.Done,
    Done    => ,
    Busy    => ,
    Error   => ,
    ErrorID =>
);

复位轴组(
    Axis      := AXIS_Z,
    bExecute  := 伺服复位.Done,
    bVirtual  := FALSE,
    bDone     => ,
    bBusy     => ,
    bError    => ,
    nErrorID  =>
);

// 报警清除逻辑
复位触发(CLK := (伺服错误状态 OR 复位请求) AND NOT 复位中);
IF 复位触发.Q THEN
    复位中 := TRUE;
    复位请求 := FALSE;
END_IF

IF 伺服复位.Done THEN
    复位中 := FALSE;
END_IF
                  
END_PROGRAM

PROGRAM AXIS_C_PRG
  VAR
    伺服使能 : Sm3_Basic.MC_Power;  (* 轴功能块实例 *)
    伺服绝对位置执行 : Sm3_Basic.MC_MoveAbsolute;
    伺服实际位置 : Sm3_Basic.MC_ReadActualPosition;
    伺服停止 : Sm3_Basic.MC_Stop;
    伺服复位 : Sm3_Basic.MC_Reset;
    伺服状态 : Sm3_Basic.MC_ReadStatus;
    复位轴组 : Sm3_Basic.SMC3_ReinitDrive;
    当前位置 : LREAL;  (* 变量 *)
    轴组复位 : BOOL;
    目标位置 : LREAL;
    目标速度 : LREAL;
    伺服错误状态 : BOOL;
    轴使能状态 : BOOL;
    总线状态 : BOOL;
    复位触发 : R_TRIG;  (* 报警清除相关 *)
    复位请求 : BOOL;
    复位中 : BOOL;
    POS_DEAD_ZONE : REAL := 0.01;  (* 死区常量 *)
    diff_old : BOOL := FALSE;  (* 上升沿检测 *)
    diff : BOOL;
    保持使能 : BOOL := FALSE;  (* 控制 MC_Power.Enable *)
    EnRise : R_TRIG;  (* 外部使能上升沿 *)
    PowerStatusRise : R_TRIG;  (* 轴使能状态上升沿 *)
    move_trigger : R_TRIG;
    AXIS_C_EXCUSE : BOOL := FALSE;
    AXIS_C_Done_Internal : BOOL;
    log_msg : STRING(100);
  END_VAR

                    //------------------------------------------------------------------
// Z 轴控制逻辑（简化版 - 仅上升沿触发）
//------------------------------------------------------------------

// 读取实际位置
伺服实际位置(
    Axis    := AXIS_C,
    Enable  := TRUE,
    Position=> 当前位置
);
GVL.Axes[5].ActualAngle := 当前位置;

// 读取轴状态
伺服状态(
    Axis    := AXIS_C,
    Enable  := TRUE,
    Valid   => ,
    Busy    => ,
    Error   => 伺服错误状态,
    ErrorID => ,
    Disabled=> 总线状态
);

// 轴使能控制
伺服使能(
    Axis               := AXIS_C,
    Enable             := TRUE,
    bRegulatorOn       := GVL.Axes[5].AxisEnable,
    bDriveStart        := GVL.Axes[5].AxisEnable,
    Status             => 轴使能状态,
    bRegulatorRealState=> ,
    bDriveStartRealState=> ,
    Busy               => ,
    Error              => ,
    ErrorID            =>
);

// 目标位置、速度赋值（来自全局变量）
目标位置 := GVL.Axes[5].TargetAngle;
目标速度 :=  GVL.Axes[5].TargetVel;

// ********** 核心：上升沿触发运动 **********
// 使用 R_TRIG 检测 need_move 的上升沿
move_trigger(CLK := GVL.Axes[5].NeedMoveAxis);
IF move_trigger.Q THEN
    AXIS_C_EXCUSE := TRUE;   // 产生一个扫描周期的脉冲
	log_msg := 'C-axis has been triggered';
// 	logfb(write:=TRUE,sFileTestString:=log_msg);
	AppendLog(log_msg);
ELSE
    AXIS_C_EXCUSE := FALSE;
END_IF

// 绝对定位指令
GVL.Axes[5].伺服绝对位置执行(
    Axis        := AXIS_C,
    Execute     := AXIS_C_EXCUSE,
    Position    := 目标位置,
    Velocity    := 目标速度,
    Acceleration:= 10000,//4000  //85000
    Deceleration:= 10000,//4000  //85000
    Jerk        := ,
    Direction   := ,
    BufferMode  := ,
    Done        => GVL.Axes[5].InitDone,
    Busy        => ,
    Active      => ,
    CommandAborted=> ,
    Error       => GVL.Axes[5].AxisError,
    ErrorID     =>
);

// 运动完成：清除 need_move 并通知状态机
IF  GVL.Axes[5].InitDone THEN
    GVL.Axes[5].NeedMoveAxis := FALSE;              // 清除运动请求
    GVL.Axes[5].AxisDone := TRUE;         // 通知状态机运动完成
	log_msg := 'B-Axis movement completed! ';
// 	logfb(write:=TRUE,sFileTestString:=log_msg);
// 	AppendLog(log_msg);
END_IF

// 复位功能块（保持不变）
伺服复位(
    Axis    := AXIS_C,
    Execute := 复位中 AND NOT 伺服复位.Done,
    Done    => ,
    Busy    => ,
    Error   => ,
    ErrorID =>
);

复位轴组(
    Axis      := AXIS_C,
    bExecute  := 伺服复位.Done,
    bVirtual  := FALSE,
    bDone     => ,
    bBusy     => ,
    bError    => ,
    nErrorID  =>
);

// 报警清除逻辑
复位触发(CLK := (伺服错误状态 OR 复位请求) AND NOT 复位中);
IF 复位触发.Q THEN
    复位中 := TRUE;
    复位请求 := FALSE;
END_IF

IF 伺服复位.Done THEN
    复位中 := FALSE;
END_IF
                  
END_PROGRAM

PROGRAM FiveDOF_Platform_PRG
  VAR
    final_angle : ARRAY[1..AXIS_COUNT] OF LREAL;  (* 最终目标 *)
    final_vel : ARRAY[1..AXIS_COUNT] OF LREAL;
    fbMove_2 : FB_5DOF_Platform_Move;  (* 功能块实例 *)
    trig_start : R_TRIG;  (* 触发边沿检测 *)
    i : INT;  (* 辅助 *)
    log_msg : STRING(255);
    logfb : Syslog_FB;
  END_VAR

                    
// --------------------------------------------------
// 主逻辑
// --------------------------------------------------
FOR i := 1 TO AXIS_COUNT BY 1 DO
    Axes[i].AxisEnable := TRUE; 
END_FOR
arAi_data[9]:=bfiveDOF_state;
// 检测外部移动指令
trig_start(CLK := Move_5Axis_Sign=1);
IF trig_start.Q THEN

	log_msg := 'five-axis platform starts moving';
// 	logfb(write:=TRUE,sFileTestString:=log_msg);
	AppendLog(log_msg);

    // 使能所有轴（可放在这里一次性使能）
	bfiveDOF_state:=1;//开始运动
    AppendLog('status 0:6-axis start move' );
    step := 10;   // 开始安全顺序
END_IF

CASE step OF
    0: // 空闲
		bfiveDOF_state:=0;//开始运动
    // ---------- 阶段1：轴移动到目标 ----------
    10:
		FOR i := 1 TO AXIS_COUNT DO
			final_angle[i] := PlatformTargetAngle[i];
			final_vel[i]   := 360*6000/60;
			Axes[i].AxisDone := FALSE;  
			GVL.Axes[i].NeedMoveAxis := TRUE;
		END_FOR
        fbMove_2(AxisAngle := final_angle, AxisVel := final_vel, Execute := TRUE,Monitor:=TRUE);
        step := 20;

		log_msg := 'State 20: Start moving XYABC AXIS... ';
// 		logfb(write:=TRUE,sFileTestString:=log_msg);
		AppendLog(log_msg);;
    20:
        fbMove_2(AxisAngle := final_angle, AxisVel := final_vel, Execute := FALSE,Monitor:=TRUE);
        IF fbMove_2.allDone THEN
			log_msg := 'State 21: XYZABC AXIS movement completed';
// 			logfb(write:=TRUE,sFileTestString:=log_msg);
			AppendLog(log_msg);
        ELSIF fbMove_2.Error THEN
            bfiveDOF_state:=2;
        END_IF
		step := 0;

        
        
END_CASE
                  
END_PROGRAM

FUNCTION_BLOCK Syslog_FB
  VAR_INPUT
    write : BOOL;
    sFileTestString : STRING(4096) := '12$N3458';
  END_VAR
  VAR
    sFileName : CAA.FILENAME := './TestFile.csv';
    first : BOOL := TRUE;
    fOpen : FILE.Open;
    fWrite : FILE.Write;
    fRead : FILE.Read;
    fClose : FILE.Close;
    hFile : CAA.HANDLE;  (* 写入 *)
    temp : INT := 0;
    t0 : ton;
    read : BOOL;  (* 读 *)
    sBuffer : STRING(4096);  (* 读取缓冲区 *)
    temp1 : INT;
    t1 : ton;
    tempWriteStr : STRING(4096);
  END_VAR

                    
IF  first THEN              //如果没有文件，将创建文件
	fOpen.sFileName := sFileName;
    fOpen.eFileMode := FILE.MODE.MWRITEPLUS;//模式选择
    fOpen(xExecute := TRUE);
	IF  fOpen.xDone THEN
		 fOpen(xExecute := FALSE);
		  first:=FALSE;
	END_IF
END_IF


//执行写入操作
// IF  write THEN  //
// 	temp:=1;
//    write:=0;	
// END_IF

CASE temp OF
	0:
		IF write THEN
			temp:=1;
		END_IF

	1:fOpen.sFileName := sFileName;
      fOpen.eFileMode := FILE.MODE.MAPPD;//模式选择
      fOpen(xExecute := TRUE);
	  t0(IN:=1 , PT:=T#5MS);
	  IF t0.Q THEN
		 temp:=2; 
         t0(IN:=0);
	  END_IF

// 	 	IF fOpen.xDone THEN
//             fOpen(xExecute:=FALSE);
//             temp := 2;
//         END_IF
	2:  fWrite.hFile := fOpen.hFile;//文件句柄
		tempWriteStr := CONCAT(sFileTestString, '$R$N');
		
		fWrite.pBuffer := ADR(tempWriteStr);
		fWrite.szSize := LEN(tempWriteStr);	
				
        fWrite(xExecute := TRUE);//写入使能
	

// 		IF fWrite.xDone THEN
//             fWrite(xExecute:=FALSE);
//             temp := 3;
//         END_IF
		t0(IN:=1 , PT:=T#5MS);
	  IF t0.Q THEN
		 temp:=3; 
         t0(IN:=0); 
	  END_IF
	3:	fClose.hFile := fOpen.hFile;//文件句柄
        fClose(xExecute := TRUE);//使能关闭文件 
		t0(IN:=1 , PT:=T#5MS);
	  IF t0.Q THEN
		 temp:=4; 
         t0(IN:=0); 
	  END_IF
	4:	fWrite(xExecute := FALSE);//写入使能
	    fClose(xExecute :=FALSE);//使能关闭文件
		fOpen(xExecute := FALSE);//打开文件使能
		 t0(IN:=1 , PT:=T#5MS);
	  IF t0.Q THEN
		 temp:=0; 
         t0(IN:=0); 
	  END_IF
END_CASE


//读取操作
IF read THEN  //
	temp1:=1;
    read:=0;	
END_IF
CASE temp1 OF
	1:fOpen.sFileName := sFileName;
      fOpen.eFileMode := FILE.MODE.MREAD;//模式选择
      fOpen(xExecute := TRUE);
	  t1(IN:=1 , PT:=T#5MS);
	  IF t1.Q THEN
		 temp1:=2; 
         t1(IN:=0);
	  END_IF
	2:  fRead.hFile := fOpen.hFile;//文件句柄
        fRead.pBuffer := ADR(sBuffer);//放到缓存区
        fRead.szBuffer := SIZEOF(sBuffer);//长度  byte
        fRead(xExecute := TRUE);
		t1(IN:=1 , PT:=T#5MS);
	  IF t1.Q THEN
		 temp1:=3; 
         t1(IN:=0); 
	  END_IF
	3:	fClose.hFile := fOpen.hFile;//文件句柄
        fClose(xExecute := TRUE);//使能关闭文件 
		t1(IN:=1 , PT:=T#5MS);
	  IF t1.Q THEN
		 temp1:=4; 
         t1(IN:=0); 
	  END_IF
	4:	 fRead(xExecute := FALSE);//写入使能
	    fClose(xExecute :=FALSE);//使能关闭文件
		fOpen(xExecute := FALSE);//打开文件使能
		 t1(IN:=1 , PT:=T#5MS);
	  IF t1.Q THEN
		 temp1:=0; 
         t1(IN:=0); 
	  END_IF
END_CASE

                  
END_FUNCTION_BLOCK

FUNCTION AppendLog : BOOL
  VAR_INPUT
    sMsg : STRING(100);
  END_VAR
  VAR
    nextHead : INT;
    pEntry : POINTER TO LogQueueEntry;
  END_VAR

                    

// 申请锁（自旋）
WHILE g_QueueLock  DO ;  END_WHILE
g_QueueLock := TRUE;

nextHead := (g_QueueHead + 1) MOD 100;
IF nextHead = g_QueueTail THEN
    // 队列满：丢弃日志（可增加丢弃计数器）
    g_QueueLock := FALSE;
//     RETURN FALSE;
END_IF

pEntry := ADR(g_LogQueue[g_QueueHead]);
pEntry^.sMsg := sMsg;
pEntry^.timestamp := TIME_TO_UDINT( TIME() );//SysTimeGetMs();   // 获取时间戳
g_QueueHead := nextHead;
g_QueueCount := g_QueueCount + 1;

g_QueueLock := FALSE;
// RETURN TRUE;
                  
END_FUNCTION

PROGRAM LogConsumer
  VAR
    entry : LogQueueEntry;
    nextTail : INT;
    pBufEntry : POINTER TO LogEntry;  (* 将日志写入 g_LogBuffer 所需临时变量 *)
    newWriteIdx : INT;
  END_VAR

                    
// 从队列取出一条日志
WHILE g_QueueLock DO ; END_WHILE
g_QueueLock := TRUE;
IF g_QueueHead = g_QueueTail THEN
    g_QueueLock := FALSE;
    RETURN;
END_IF

entry := g_LogQueue[g_QueueTail];
nextTail := (g_QueueTail + 1) MOD 100;
g_QueueTail := nextTail;
g_QueueCount := g_QueueCount - 1;
g_QueueLock := FALSE;

// --- 以下将 entry 写入环形缓冲区 g_LogBuffer（单线程，无需锁）---
// 注意：这里直接操作 g_LogBuffer，与 Modbus 映射代码共享
// 但 Modbus 映射代码只读，不会写，所以安全
// 但需要确保 Modbus 映射读取时不会读到一半更新的条目（可以通过双缓冲或版本号避免，但通常可以接受）

newWriteIdx := (g_LogBuffer.writeIdx + 1) MOD g_LogBuffer.maxSize;
IF newWriteIdx = g_LogBuffer.readIdx THEN
    // 缓冲区满，覆盖最旧
    g_LogBuffer.readIdx := (g_LogBuffer.readIdx + 1) MOD g_LogBuffer.maxSize;
    // count 不变
ELSE
    g_LogBuffer.count := g_LogBuffer.count + 1;
END_IF

pBufEntry := ADR(g_LogBuffer.entries[g_LogBuffer.writeIdx]);
pBufEntry^.sMessage := entry.sMsg;
pBufEntry^.length := LEN(entry.sMsg);
pBufEntry^.timestamp := entry.timestamp;
g_LogBuffer.writeIdx := newWriteIdx;
                  
END_PROGRAM

PROGRAM JogY
  VAR
    fbJogX : FB_ServoJog;
    fbJogY : FB_ServoJog;
    fbJogZ : FB_ServoJog;
    fbJogB : FB_ServoJog;
    fbJogC : FB_ServoJog;
    xServoEnable : BOOL := TRUE;
  END_VAR

                    

 




  // ================================
  // 5轴点动控制
  // ================================


  fbJogY(
      Axis := AXIS_Y,
      xServoOn := xServoEnable,
      xReset := FALSE,
      xJogFwd := xJogFwd[2],
      xJogRev := xJogRev[2],
      xLimitFwd := FALSE,
      xLimitRev := FALSE,
      lrJogVel := 100.0,
      lrAcc := 100.0,
      lrDec := 200.0,
      lrJerk := 0.0
  );

 
                  
END_PROGRAM

FUNCTION_BLOCK FB_ServoJog
  VAR_IN_OUT
    Axis : AXIS_REF_SM3;  (* 设备树中的伺服轴 *)
  END_VAR
  VAR_INPUT
    xServoOn : BOOL;  (* 伺服使能 *)
    xReset : BOOL;  (* 故障复位按钮 *)
    xJogFwd : BOOL;  (* 正向点动按钮 *)
    xJogRev : BOOL;  (* 反向点动按钮 *)
    xLimitFwd : BOOL;  (* 正限位，TRUE = 已触发 *)
    xLimitRev : BOOL;  (* 负限位，TRUE = 已触发 *)
    lrJogVel : LREAL := 100.0;  (* 点动速度 *)
    lrAcc : LREAL := 100.0;  (* 加速度 *)
    lrDec : LREAL := 100.0;  (* 减速度 *)
    lrJerk : LREAL := 0.0;  (* 加加速度，0 表示不用 *)
  END_VAR
  VAR_OUTPUT
    xReady : BOOL;  (* 伺服已上使能 *)
    xMoving : BOOL;  (* 正在点动 *)
    xFault : BOOL;  (* 程序/运动控制故障 *)
    iFaultSrc : INT;  (* 0无故障，1Power，2Reset，3Jog，10方向按钮冲突 *)
  END_VAR
  VAR
    fbPower : MC_Power;
    fbReset : MC_Reset;
    fbJog : MC_Jog;
    rtReset : R_TRIG;
    xCmdFwd : BOOL;
    xCmdRev : BOOL;
    xConflict : BOOL;
  END_VAR
  VAR_OUTPUT
    xJogFwdCmd : BOOL;
    xJogRevCmd : BOOL;
    xJogError : BOOL;
    eJogErrorID : SMC_ERROR;
    xJogAborted : BOOL;
  END_VAR

                     
 // 伺服上使能
  fbPower(
      Axis :=Axis,
      Enable := xServoOn,
      bRegulatorOn := TRUE,
      bDriveStart := TRUE
  );

 
  // 故障复位，上升沿触发
  rtReset(CLK := xReset);

  fbReset(
      Axis :=Axis,
      Execute := rtReset.Q
  );

  // 防止正反同时点动
  xConflict := xJogFwd AND xJogRev;

  // 点动允许条件
  xCmdFwd := xJogFwd
             AND  fbPower.Status
            AND NOT xJogRev
             AND NOT xLimitFwd
            AND NOT xConflict;

  xCmdRev := fbPower.Status
             AND xJogRev
             AND NOT xJogFwd
             AND NOT xLimitRev
             AND NOT xConflict;

  // 点动控制：按住走，松开按减速度停止
  fbJog(
      Axis := Axis,
      JogForward := xCmdFwd,
      JogBackward := xCmdRev,
      Velocity := lrJogVel,
      Acceleration := lrAcc,
      Deceleration := lrDec,
      Jerk := lrJerk
  );

  // 状态输出
  xReady := fbPower.Status;
  xMoving := fbJog.Busy;

  xFault := fbPower.Error OR fbReset.Error OR fbJog.Error OR xConflict;

  IF fbPower.Error THEN
      iFaultSrc := 1;
  ELSIF fbReset.Error THEN
      iFaultSrc := 2;
  ELSIF fbJog.Error THEN
      iFaultSrc := 3;
  ELSIF xConflict THEN
      iFaultSrc := 10;
  ELSE
      iFaultSrc := 0;
  END_IF;
  
  xJogFwdCmd := xCmdFwd;
  xJogRevCmd := xCmdRev;
  xJogError := fbJog.Error;
  eJogErrorID := fbJog.ErrorID;
  xJogAborted := fbJog.CommandAborted;

 
                  
END_FUNCTION_BLOCK

PROGRAM JogX
  VAR
    fbJogX : FB_ServoJog;
    xServoEnable : BOOL := TRUE;
  END_VAR

                    

 



 xJogMode[1] := (arReg_data[19] AND WORD#16#0001) <> WORD#0; // X
 
  // ================================
  // 5轴点动控制
  // ================================

  fbJogX(
      Axis := AXIS_X,
      xServoOn := xServoEnable,
      xReset := FALSE,
      xJogFwd := xJogFwd[1],
      xJogRev := xJogRev[1],
      xLimitFwd := FALSE,
      xLimitRev := FALSE,
      lrJogVel := 100.0,
      lrAcc := 100.0,
      lrDec := 200.0,
      lrJerk := 0.0
  );

                  
END_PROGRAM

PROGRAM JogB
  VAR
    fbJogX : FB_ServoJog;
    fbJogY : FB_ServoJog;
    fbJogZ : FB_ServoJog;
    fbJogB : FB_ServoJog;
    fbJogC : FB_ServoJog;
    xServoEnable : BOOL := TRUE;
  END_VAR

                    

 




  // ================================
  // 5轴点动控制
  // ================================

  
  fbJogB(
      Axis := AXIS_B,
      xServoOn := xServoEnable,
      xReset := FALSE,
      xJogFwd := xJogFwd[4],
      xJogRev := xJogRev[4],
      xLimitFwd := FALSE,
      xLimitRev := FALSE,
      lrJogVel := 100.0,
      lrAcc := 100.0,
      lrDec := 200.0,
      lrJerk := 0.0
  );

 
                  
END_PROGRAM

PROGRAM JogZ
  VAR
    fbJogX : FB_ServoJog;
    fbJogY : FB_ServoJog;
    fbJogZ : FB_ServoJog;
    fbJogB : FB_ServoJog;
    fbJogC : FB_ServoJog;
    xServoEnable : BOOL := TRUE;
  END_VAR

                    

 




  // ================================
  // 5轴点动控制
  // ================================

  

  fbJogZ(
      Axis := AXIS_Z,
      xServoOn := xServoEnable,
      xReset := FALSE,
      xJogFwd := xJogFwd[3],
      xJogRev := xJogRev[3],
      xLimitFwd := FALSE,
      xLimitRev := FALSE,
      lrJogVel := 100.0,
      lrAcc := 100.0,
      lrDec := 200.0,
      lrJerk := 0.0
  );

 
                  
END_PROGRAM

PROGRAM JogC
  VAR
    fbJogX : FB_ServoJog;
    fbJogY : FB_ServoJog;
    fbJogZ : FB_ServoJog;
    fbJogB : FB_ServoJog;
    fbJogC : FB_ServoJog;
    xServoEnable : BOOL := TRUE;
  END_VAR

                    

 




  // ================================
  // 5轴点动控制
  // ================================

  fbJogC(
      Axis := AXIS_C,
      xServoOn := xServoEnable,
      xReset := FALSE,
      xJogFwd := xJogFwd[5],
      xJogRev := xJogRev[5],
      xLimitFwd := FALSE,
      xLimitRev := FALSE,
      lrJogVel := 100.0,
      lrAcc := 100.0,
      lrDec := 200.0,
      lrJerk := 0.0
  );
                  
END_PROGRAM

CONFIGURATION Device
  RESOURCE Application ON PLC
    VAR_GLOBAL CONSTANT  (* GVL *)
      AXIS_COUNT : INT := 5;
      使能 : BOOL;  (* 接收到的目标角度（浮点数） *)
      Axes : ARRAY[1..5] OF Axis;  (* 5个轴的结构体数组 *)
      Move_5Axis_Sign : INT;
      step : INT := 0;  (* 0空闲, 10平台运动 20运动完成 *)
      bModeSwitchDone : BOOL := FALSE;
      torque_pos_change : BOOL := TRUE;
      PlatformTargetAngle : ARRAY[1..AXIS_COUNT] OF LREAL;
      PlatformTargetVel : ARRAY[1..AXIS_COUNT] OF LREAL;
      pushmotorpos : LREAL;
      arDo_data : ARRAY[0..16] OF BOOL;  (* 用于存放线圈的数据 *)
      arDi_data : ARRAY[0..15] OF BOOL;  (* 用于存放离散型数据 *)
      arReg_data : ARRAY[0..199] OF INT;  (* 用于存放保持型寄存器的数据 *)
      arAi_data : ARRAY[0..16] OF INT;  (* 用于存放输入型寄存器的数据 *)
      mchome : Sm3_Basic.MC_Home;
      DoorlockHomedone : BOOL;
      StrikeplateHomedone : BOOL;
      bfiveDOF_state : INT;
      xJogFwd : ARRAY[1..5] OF BOOL;
      xJogRev : ARRAY[1..5] OF BOOL;
      xJogMode : ARRAY[1..5] OF BOOL;
      g_LogBuffer : LogBuffer := (writeIdx := 0, readIdx := 0, count := 0, maxSize := 10);  (* 日志modbus 日志缓冲区配置 *)
      g_bLogNew : BOOL;  (* 可选：有新日志标志（供主站快速判断） *)
      g_LogLock : BOOL := FALSE;  (* 互斥标志 *)
      g_LogQueue : ARRAY[0..199] OF LogQueueEntry;  (* 增大队列深度 *)
      g_QueueHead : INT := 0;
      g_QueueTail : INT := 0;
      g_QueueCount : INT := 0;
      g_QueueLock : BOOL := FALSE;
    END_VAR
    TASK EtherCAT_Task(INTERVAL := T#4ms, PRIORITY := 1);
    TASK MainTask(INTERVAL := T#5ms, PRIORITY := 1);
    PROGRAM JogX WITH EtherCAT_Task : JogX;
    PROGRAM JogY WITH EtherCAT_Task : JogY;
    PROGRAM JogZ WITH EtherCAT_Task : JogZ;
    PROGRAM JogB WITH EtherCAT_Task : JogB;
    PROGRAM JogC WITH EtherCAT_Task : JogC;
    PROGRAM AXIS_X_PRG WITH EtherCAT_Task : AXIS_X_PRG;
    PROGRAM Axis_Y_PRG WITH EtherCAT_Task : Axis_Y_PRG;
    PROGRAM AXIS_Z_PRG WITH EtherCAT_Task : AXIS_Z_PRG;
    PROGRAM AXIS_B_PRG WITH EtherCAT_Task : AXIS_B_PRG;
    PROGRAM AXIS_C_PRG WITH EtherCAT_Task : AXIS_C_PRG;
    PROGRAM FiveDOF_Platform_PRG WITH MainTask : FiveDOF_Platform_PRG;
    PROGRAM LogConsumer WITH MainTask : LogConsumer;
    PROGRAM PLC_PRG WITH MainTask : PLC_PRG;
    PROGRAM AxisStatusFeedback_PRG WITH MainTask : AxisStatusFeedback_PRG;
    PROGRAM ModbusTcpSlave WITH MainTask : ModbusTcpSlave;
  END_RESOURCE
END_CONFIGURATION

CONFIGURATION EtherCAT_Master_SoftMotion
END_CONFIGURATION

CONFIGURATION LC10E_V1_04
END_CONFIGURATION

CONFIGURATION AXIS_X
END_CONFIGURATION

CONFIGURATION LC10E_V1_04_1
END_CONFIGURATION

CONFIGURATION AXIS_Y
END_CONFIGURATION

CONFIGURATION LC10E_V1_04_4
END_CONFIGURATION

CONFIGURATION AXIS_Z
END_CONFIGURATION

CONFIGURATION LC10E_V1_04_6
END_CONFIGURATION

CONFIGURATION AXIS_B
END_CONFIGURATION

CONFIGURATION LC10E_V1_04_7
END_CONFIGURATION

CONFIGURATION AXIS_C
END_CONFIGURATION

CONFIGURATION SoftMotion General Axis Pool
END_CONFIGURATION
